Fanuc KAREL source: kt00126.KL

-- PROVISIONAL review KL for V940-1; original PC SHA256 696e7c321af5a132be7241e874939ecfa48c1ee9b9852a1db1c623146b45b15d
-- Incomplete behavior may be omitted. Consult companion uncertainty JSON. Do not deploy.
PROGRAM KT00126
%NOLOCKGROUP
VAR
  OUT : REAL
-- UNRESOLVED_DECL H1 type=002017
-- UNRESOLVED_DECL Y2 type=002018
BEGIN
  -- V9_ZERO_TABLE_METADATA_HINT layout=0001; no indexed target words; source/name/runtime held
  -- UNRESOLVED_PC offsets 5-19; opcodes 2E,22,9D,33,B4
  -- UNRESOLVED_PC offsets 24-38; opcodes 2E,22,9D,33,B2
  -- UNRESOLVED_PC offsets 43-72; opcodes 22,9D,33,B3,22,9D,33,B1,64,29,64,29,6C,23
  -- UNRESOLVED_PC offsets 77-81; opcodes 7F
END KT00126
